{attribute addProperty BoxType "KL2212"}
{attribute addProperty Id "WireBreakAT %I*BOOL000CurcuitAT %I*BOOL000OutputAT %Q*BOOL000"}
{attribute addProperty CRC "2437386886"}
{attribute addProperty SizeInBites "0"}
{attribute addProperty SizeInBytes "0"}
TYPE Channel_91479286 :
STRUCT
	{attribute addProperty Name "WireBreak"}
	WireBreak AT %I* : BOOL;
	{attribute addProperty Name "Curcuit"}
	Curcuit AT %I* : BOOL;
	{attribute addProperty Name "Output"}
	Output AT %Q* : BOOL;
END_STRUCT
END_TYPE

(* stored: Version 1.2.0.0, ProductVersion 3.1.4024.9
   DUT Channel_91479286: Id {5bcab5f1-d6a5-4f47-8f48-f10c67c3a9c7} *)
